{attribute 'linkalways'} 
{attribute 'no_explicit_call' := 'This FB is a CLASS and must be accessed using methods or properties'}
{attribute 'enable_dynamic_creation'}
FUNCTION_BLOCK _ETcVnStructuringElementShape EXTENDS EnumDatatypeBase
VAR
	localData : ETcVnStructuringElementShape;
	activeData : REFERENCE TO ETcVnStructuringElementShape;
	enumBaseDatatype : _DINT(localData);
END_VAR

METHOD PRIVATE AddLocalEnumeration
VAR_INPUT
	Enumeration : T_MAXSTRING;
	Value : ETcVnStructuringElementShape;
END_VAR
AddEnumeration(Enumeration, Value);
END_METHOD

PROPERTY PUBLIC Address : PVOID
GET
Address := ADR(activeData);
END_GET
END_PROPERTY

METHOD PUBLIC ClearReference
VAR_INPUT
END_VAR
activeData REF= localData;
SetBaseDatatypeReference();
END_METHOD

METHOD PUBLIC Clone : I_Datatype
VAR
    pClone : POINTER TO _ETcVnStructuringElementShape;
END_VAR
pClone := __NEW(_ETcVnStructuringElementShape(InitialValue := Value));
Clone := pClone^;
END_METHOD

METHOD FB_init : BOOL
VAR_INPUT
	bInitRetains : BOOL; // if TRUE, the retain variables are initialized (warm start / cold start)
	bInCopyCode : BOOL;  // if TRUE, the instance afterwards gets moved into the copy code (online change)
	InitialValue : ETcVnStructuringElementShape;
END_VAR
localData := InitialValue;
AddBaseDatatype(enumBaseDatatype);
ClearReference();

AddLocalEnumeration('TCVN_SES_RECTANGLE', ETcVnStructuringElementShape.TCVN_SES_RECTANGLE);
AddLocalEnumeration('TCVN_SES_CROSS', ETcVnStructuringElementShape.TCVN_SES_CROSS);
AddLocalEnumeration('TCVN_SES_ELLIPSE', ETcVnStructuringElementShape.TCVN_SES_ELLIPSE);
END_METHOD

PROPERTY PUBLIC Identifier : T_MAXSTRING
GET
Identifier := 'ETcVnStructuringElementShape';
END_GET
END_PROPERTY

METHOD IsEnumeratorValueEqual : BOOL
VAR_INPUT
	Enumerator : I_KeyValueForwardEnumerator;
END_VAR
VAR
	storedValue : ETcVnStructuringElementShape;
END_VAR
IF NOT Enumerator.TryGet(storedValue) THEN
	RETURN;
END_IF

IsEnumeratorValueEqual := storedValue = activeData;
END_METHOD

METHOD PUBLIC MakeReferenceTo
VAR_INPUT
	ReferenceTarget : REFERENCE TO ETcVnStructuringElementShape;
END_VAR
activeData REF= ReferenceTarget;
SetBaseDatatypeReference();
END_METHOD

METHOD PROTECTED SetBaseDatatypeReference
VAR_INPUT
END_VAR
enumBaseDatatype.MakeReferenceTo(activeData);
END_METHOD

PROPERTY PUBLIC Size : UDINT
GET
Size := SIZEOF(activeData);
END_GET
END_PROPERTY

METHOD TryMakeReferenceTo : BOOL
VAR_INPUT
	Target : I_Datatype;
END_VAR
VAR
	targetAsEnum : I_EnumDatatype;
	pTargetData : POINTER TO ETcVnStructuringElementShape;
END_VAR
IF NOT Target.TryResolveAsEnumDatatype(targetAsEnum) THEN
	RETURN;
END_IF

IF targetAsEnum.Identifier <> Identifier THEN
	RETURN;
END_IF

pTargetData := Target.Address;
activeData REF= pTargetData^;
SetBaseDatatypeReference();
TryMakeReferenceTo := TRUE;
END_METHOD

PROPERTY PUBLIC Value : ETcVnStructuringElementShape
GET
Value := activeData;
END_GET
SET
activeData := Value;
END_SET
END_PROPERTY

END_FUNCTION_BLOCK

(* stored: Version 1.1.0.1
   POU _ETcVnStructuringElementShape: Id {2371b4b7-6374-459e-9198-e8d5fc834d5b}, SpecialFunc None
   Folder Constructor: Id {0acb9418-4d56-4db7-a073-44a801102ebb}
   Folder Private: Id {7023aef0-49a3-4da0-aa7e-4739a1bdc889}
   Folder Protected: Id {6fb0cd12-812e-4218-90af-756e5ff9ccfb}
   Method AddLocalEnumeration: Id {e708d138-1c71-4fa0-9e94-7533385ecbfc}
   Property Address: Id {d3e551ee-eab7-4b35-b2f5-786567f673a7}
   Get Get: Id {cbd37d27-2edb-4149-86aa-c25c58cd59ff}
   Method ClearReference: Id {51b447d2-f3a9-4371-b528-289d2004c08b}
   Method Clone: Id {c42ae7f8-5f8a-4438-87e9-22d2152f9624}
   Method FB_init: Id {9db52dcd-a29d-42be-8f8c-360d9c7f7f18}
   Property Identifier: Id {a7497406-b61e-4a4d-bac0-54091b3148b8}
   Get Get: Id {ca454450-e8aa-4450-b26d-8e877e4b0b16}
   Method IsEnumeratorValueEqual: Id {18a039d3-376a-4cfb-94e2-8d2e3cf1107e}
   Method MakeReferenceTo: Id {e90b1cfd-e4a4-4f00-a6d5-ace1e300e352}
   Method SetBaseDatatypeReference: Id {f6ac004b-d5ce-4f41-a51a-389c8e106294}
   Property Size: Id {3447659c-4bad-42c6-b367-b8a12dbb4a6a}
   Get Get: Id {c51fa3c0-eeb2-4e29-ba33-e4dad8162ef1}
   Method TryMakeReferenceTo: Id {c92eb8b4-f9e6-40ce-844a-44c3ca417ba8}
   Property Value: Id {3a2c52dd-83d8-43fa-968b-4bdcdb76c07c}
   Get Get: Id {c0ccde93-fc61-43ae-8070-59920d58bd34}
   Set Set: Id {ea194220-51b0-420e-9b79-99cb3aa091de} *)
